TYPE ST_ParamFixed :
STRUCT
END_STRUCT
END_TYPE

(* stored: Version 1.1.0.1, ProductVersion 3.1.4020.6
   DUT ST_ParamFixed: Id {df57b0b8-2738-4746-9062-2ea57719fdde} *)
